# EPICS autosave request: CARSApp/Db/IDD_DAC_detector_settings.req
$(P)$(T)NumPoints
$(P)$(T)TotalTime
$(P)$(T)T2Start
$(P)$(T)T2End
$(P)$(T)SDStart
$(P)$(T)SDEnd
$(P)$(T)XOStart
$(P)$(T)XOEnd
